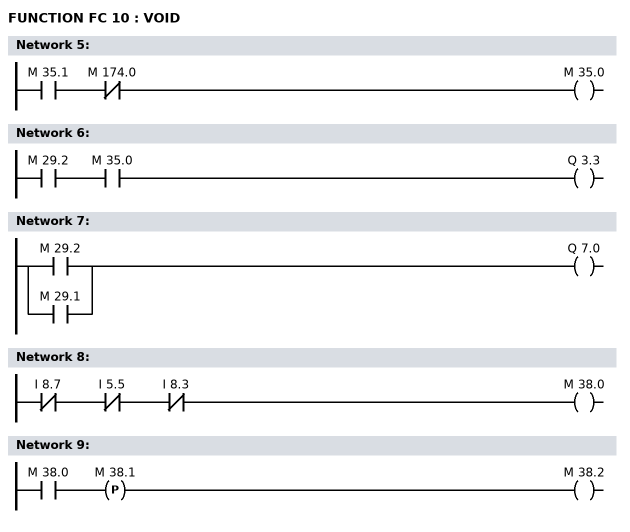

      A     M     35.1;
      AN    M    174.0;
      =     M     35.0;
NETWORK
TITLE =

      A     M     29.2;
      A     M     35.0;
      =     Q      3.3;
NETWORK
TITLE =

      O     M     29.2;
      O     M     29.1;
      =     Q      7.0;
NETWORK
TITLE =

      AN    I      8.7;
      AN    I      5.5;
      AN    I      8.3;
      =     M     38.0;
NETWORK
TITLE =

      A     M     38.0;
      FP    M     38.1;
      =     M     38.2;
NETWORK
TITLE =

      A     I      8.7;
      A(    ;
      A     I      5.5;
      L     DB2.DBW   46;
      SF    T     23;
      NOP   0;
      NOP   0;
      NOP   0;
      A     T     23;
      )     ;
      A     I      8.3;
      A     I     11.4;
      A     I     12.5;
      =     L      1.0;
      A     L      1.0;
      BLD   102;
      =     M     38.3;
      A     L      1.0;
      A     M     44.1;
      S     Q      3.5;
      A(    ;
      ON    M     44.1;
      O     ;
      A     I      0.6;
      AN    I      1.1;
      O     ;
      A     I      0.7;
      AN    I      4.1;
      )     ;
      R     Q      3.5;
      NOP   0;
NETWORK
TITLE =

      A(    ;
      A     M     35.0;
      A     #TEMP0;
      AN    #TEMP1;
      AN    M     38.3;
      FP    M     29.5;
      =     M     44.0;
      A     M     44.0;
      S     M     44.1;
      A(    ;
      O     M     20.7;
      ON    M     35.1;
      O     M     11.1;
      O     M     38.2;
      O     #TEMP1;
      O     M    114.0;
      )     ;
      R     M     44.1;
      A     M     44.1;
      )     ;
      A     M     38.3;
      O     ;
      AN    M     38.3;
      A     M     44.1;
      A     M     10.6;
      O     I      1.3;
      =     Q      3.1;
NETWORK
TITLE =
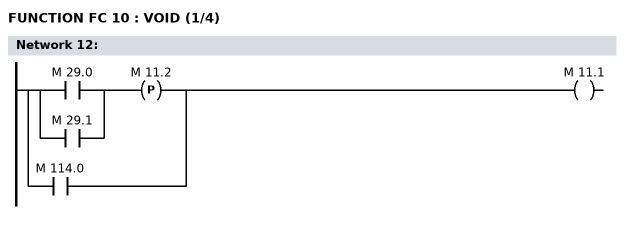

      A(    ;
      O     M     29.0;
      O     M     29.1;
      )     ;
      FP    M     11.2;
      O     M    114.0;
      =     M     11.1;
NETWORK
TITLE =
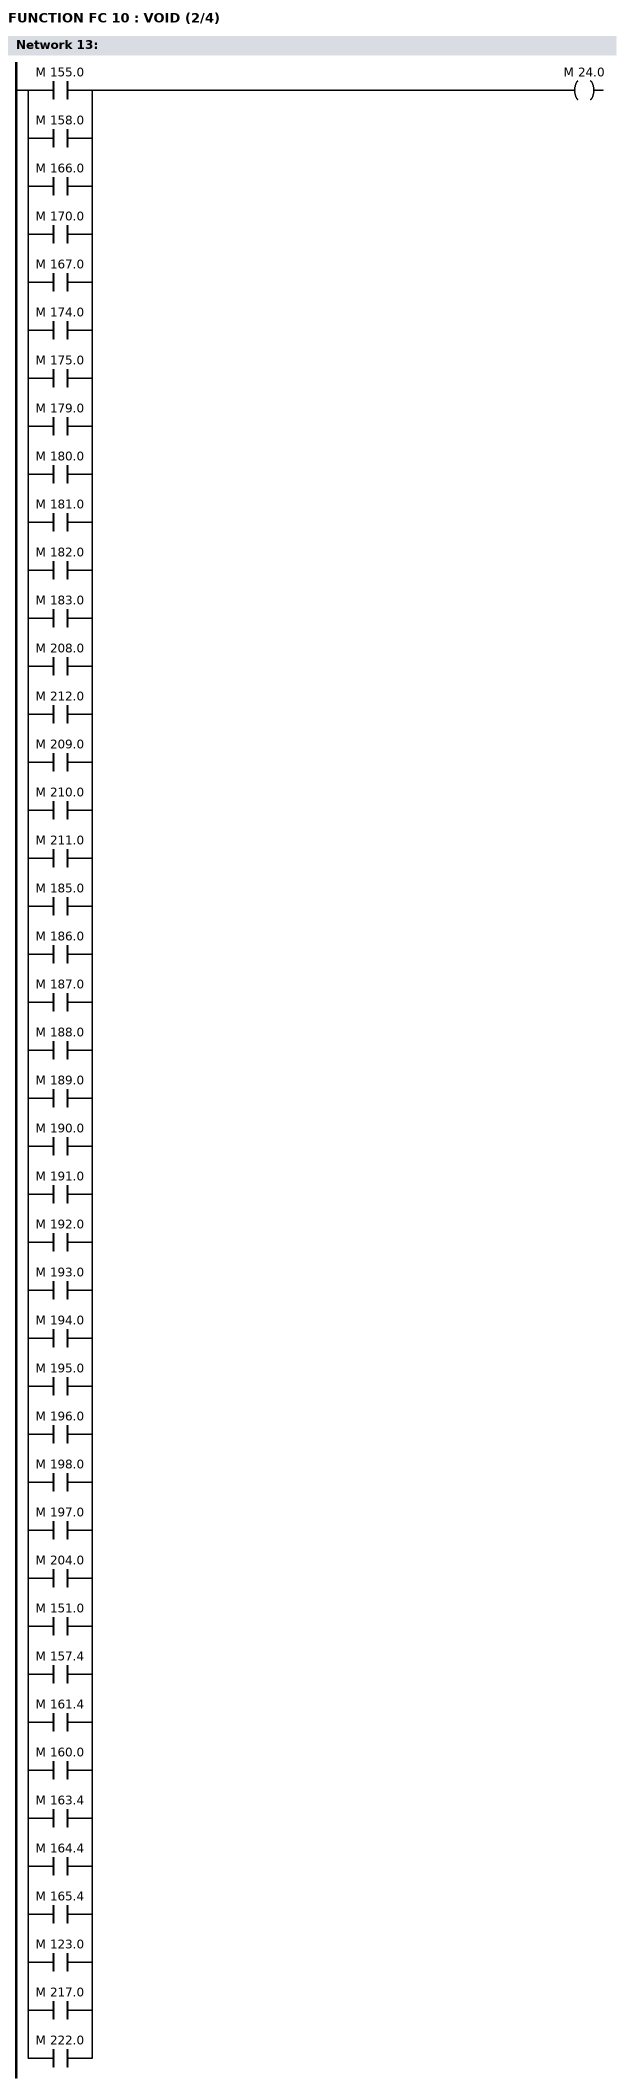

      O     M    155.0;
      O     M    158.0;
      O     M    166.0;
      O     M    170.0;
      O     M    167.0;
      O     M    174.0;
      O     M    175.0;
      O     M    179.0;
      O     M    180.0;
      O     M    181.0;
      O     M    182.0;
      O     M    183.0;
      O     M    208.0;
      O     M    212.0;
      O     M    209.0;
      O     M    210.0;
      O     M    211.0;
      O     M    185.0;
      O     M    186.0;
      O     M    187.0;
      O     M    188.0;
      O     M    189.0;
      O     M    190.0;
      O     M    191.0;
      O     M    192.0;
      O     M    193.0;
      O     M    194.0;
      O     M    195.0;
      O     M    196.0;
      O     M    198.0;
      O     M    197.0;
      O     M    204.0;
      O     M    151.0;
      O     M    157.4;
      O     M    161.4;
      O     M    160.0;
      O     M    163.4;
      O     M    164.4;
      O     M    165.4;
      O     M    123.0;
      O     M    217.0;
      O     M    222.0;
      =     M     24.0;
NETWORK
TITLE =
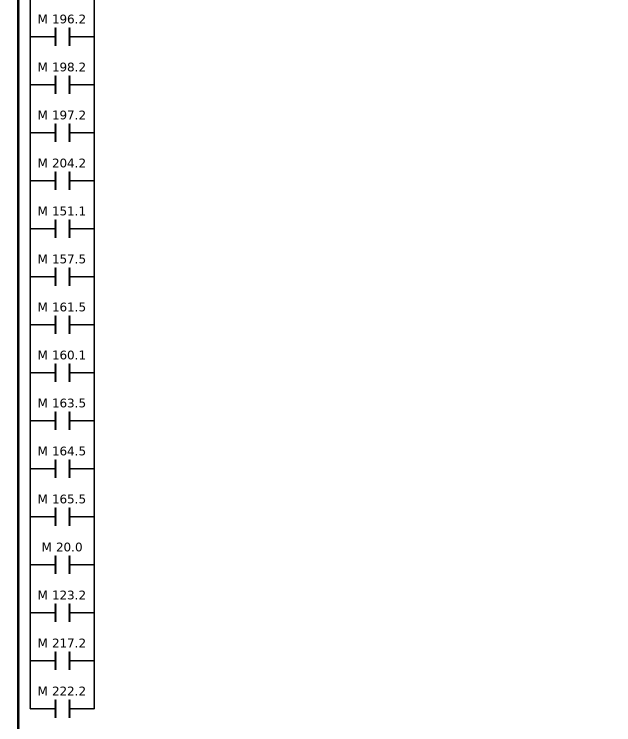

      O     M    155.2;
      O     M    158.2;
      O     M    166.2;
      O     M    170.2;
      O     M    167.2;
      O     M    174.2;
      O     M    175.2;
      O     M    179.2;
      O     M    180.2;
      O     M    181.2;
      O     M    182.2;
      O     M    183.2;
      O     M    208.2;
      O     M    212.2;
      O     M    209.2;
      O     M    210.2;
      O     M    211.2;
      O     M    185.2;
      O     M    186.2;
      O     M    187.2;
      O     M    188.2;
      O     M    189.2;
      O     M    190.2;
      O     M    191.2;
      O     M    192.2;
      O     M    193.2;
      O     M    194.2;
      O     M    195.2;
      O     M    196.2;
      O     M    198.2;
      O     M    197.2;
      O     M    204.2;
      O     M    151.1;
      O     M    157.5;
      O     M    161.5;
      O     M    160.1;
      O     M    163.5;
      O     M    164.5;
      O     M    165.5;
      O     M     20.0;
      O     M    123.2;
      O     M    217.2;
      O     M    222.2;
      =     M     22.0;
NETWORK
TITLE =
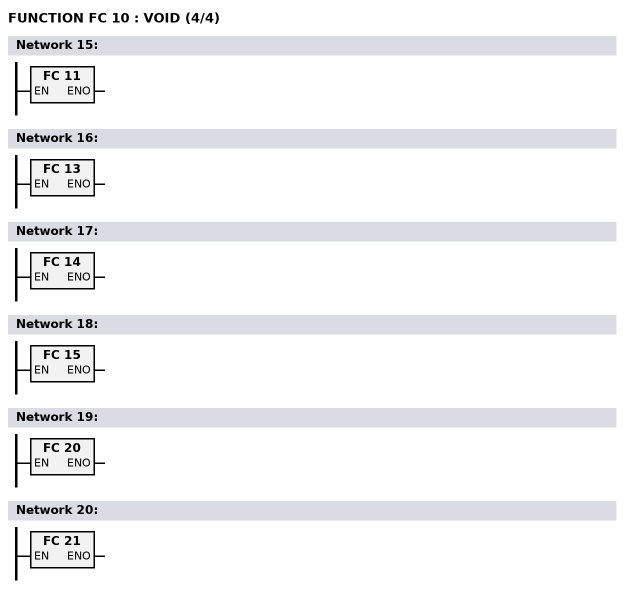

      CALL FC    11 ;
      NOP   0;
NETWORK
TITLE =

      CALL FC    13 ;
      NOP   0;
NETWORK
TITLE =

      CALL FC    14 ;
      NOP   0;
NETWORK
TITLE =

      CALL FC    15 ;
      NOP   0;
NETWORK
TITLE =

      CALL FC    20 ;
      NOP   0;
NETWORK
TITLE =

      CALL FC    21 ;
      NOP   0;
END_FUNCTION

FUNCTION FC 191 : VOID
AUTHOR :
FAMILY : ZEITEN
NAME : S_EVERZ
VERSION : 0.0


VAR_INPUT
  IN0 : BOOL ;
  IN1 : BOOL ;
END_VAR
VAR_IN_OUT
  IO2 : INT ;
  IO3 : INT ;
  IO4 : INT ;
  IO5 : INT ;
  IO6 : INT ;
  IO7 : WORD ;
END_VAR
VAR_TEMP
  TEMP8 : BOOL ;
  TEMP9 : BOOL ;
  TEMP10 : BOOL ;
  TEMP11 : BOOL ;
  TEMP12 : BOOL ;
END_VAR
BEGIN
NETWORK
TITLE =
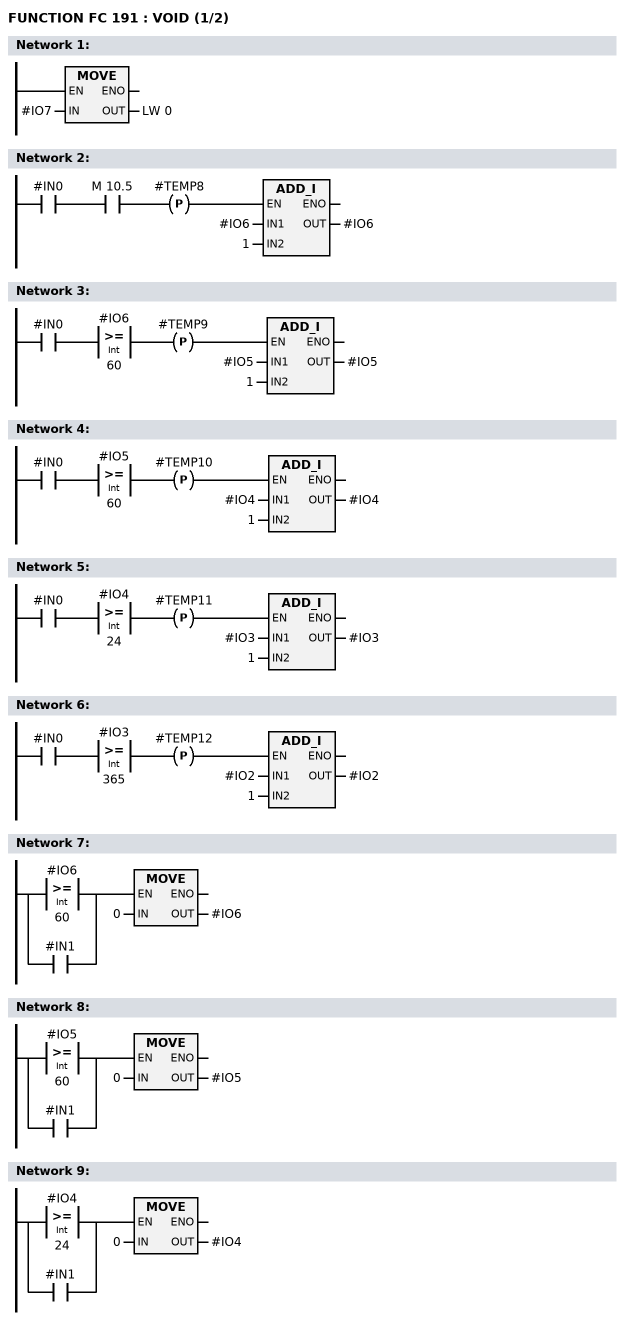

      L     #IO7;
      T     LW     0;
      NOP   0;
NETWORK
TITLE =

      A     #IN0;
      A     M     10.5;
      FP    #TEMP8;
      JNB   M001;
      L     #IO6;
      L     1;
      +I    ;
      T     #IO6;
M001: NOP   0;
NETWORK
TITLE =

      A     #IN0;
      A(    ;
      L     #IO6;
      L     60;
      >=I   ;
      )     ;
      FP    #TEMP9;
      JNB   M002;
      L     #IO5;
      L     1;
      +I    ;
      T     #IO5;
M002: NOP   0;
NETWORK
TITLE =

      A     #IN0;
      A(    ;
      L     #IO5;
      L     60;
      >=I   ;
      )     ;
      FP    #TEMP10;
      JNB   M003;
      L     #IO4;
      L     1;
      +I    ;
      T     #IO4;
M003: NOP   0;
NETWORK
TITLE =

      A     #IN0;
      A(    ;
      L     #IO4;
      L     24;
      >=I   ;
      )     ;
      FP    #TEMP11;
      JNB   M004;
      L     #IO3;
      L     1;
      +I    ;
      T     #IO3;
M004: NOP   0;
NETWORK
TITLE =

      A     #IN0;
      A(    ;
      L     #IO3;
      L     365;
      >=I   ;
      )     ;
      FP    #TEMP12;
      JNB   M005;
      L     #IO2;
      L     1;
      +I    ;
      T     #IO2;
M005: NOP   0;
NETWORK
TITLE =

      A(    ;
      O(    ;
      L     #IO6;
      L     60;
      >=I   ;
      )     ;
      O     #IN1;
      )     ;
      JNB   M006;
      L     0;
      T     #IO6;
M006: NOP   0;
NETWORK
TITLE =

      A(    ;
      O(    ;
      L     #IO5;
      L     60;
      >=I   ;
      )     ;
      O     #IN1;
      )     ;
      JNB   M007;
      L     0;
      T     #IO5;
M007: NOP   0;
NETWORK
TITLE =

      A(    ;
      O(    ;
      L     #IO4;
      L     24;
      >=I   ;
      )     ;
      O     #IN1;
      )     ;
      JNB   M008;
      L     0;
      T     #IO4;
M008: NOP   0;
NETWORK
TITLE =
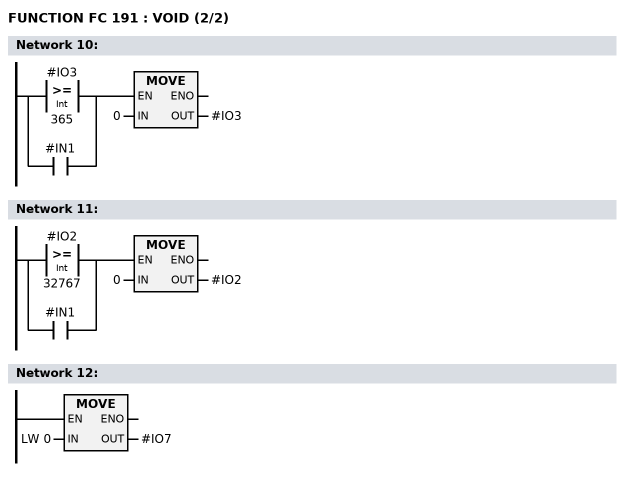

      A(    ;
      O(    ;
      L     #IO3;
      L     365;
      >=I   ;
      )     ;
      O     #IN1;
      )     ;
      JNB   M009;
      L     0;
      T     #IO3;
M009: NOP   0;
NETWORK
TITLE =

      A(    ;
      O(    ;
      L     #IO2;
      L     32767;
      >=I   ;
      )     ;
      O     #IN1;
      )     ;
      JNB   M00a;
      L     0;
      T     #IO2;
M00a: NOP   0;
NETWORK
TITLE =

      L     LW     0;
      T     #IO7;
      NOP   0;
END_FUNCTION

FUNCTION FC 1 : VOID
AUTHOR :
FAMILY : GENERAL
NAME : GENERAL
VERSION : 0.0

BEGIN
NETWORK
TITLE =
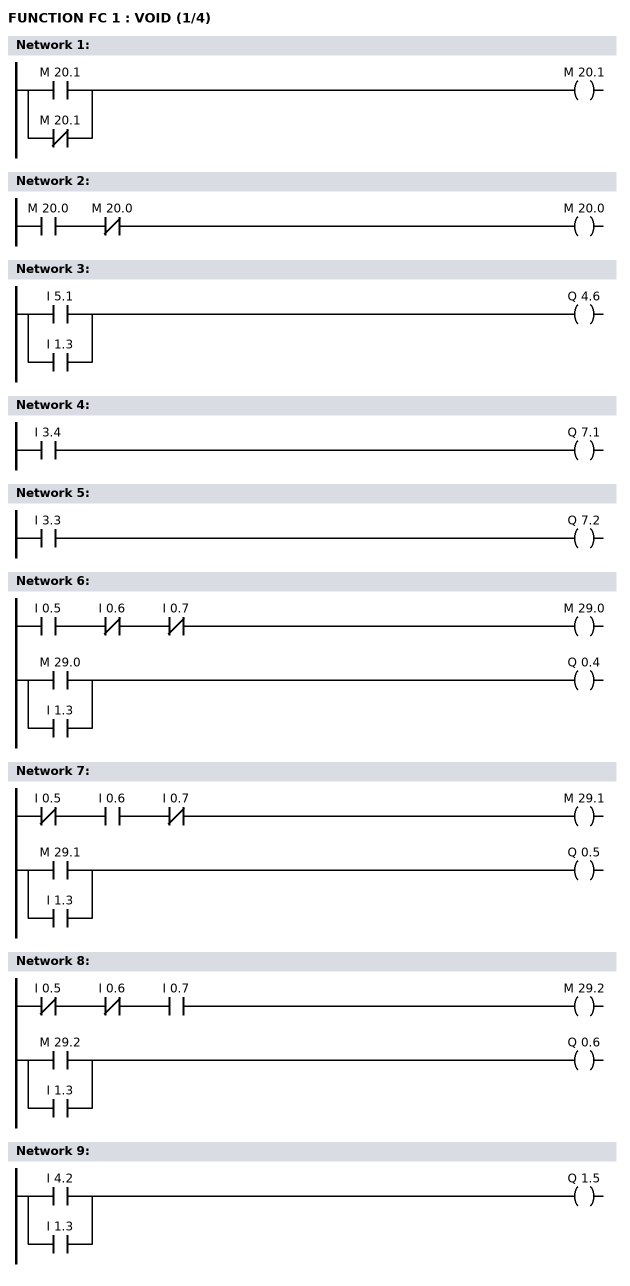

      O     M     20.1;
      ON    M     20.1;
      =     M     20.1;
NETWORK
TITLE =

      A     M     20.0;
      AN    M     20.0;
      =     M     20.0;
NETWORK
TITLE =

      O     I      5.1;
      O     I      1.3;
      =     Q      4.6;
NETWORK
TITLE =

      A     I      3.4;
      =     Q      7.1;
NETWORK
TITLE =

      A     I      3.3;
      =     Q      7.2;
NETWORK
TITLE =

      A     I      0.5;
      AN    I      0.6;
      AN    I      0.7;
      =     M     29.0;
      A     M     29.0;
      O     I      1.3;
      =     Q      0.4;
NETWORK
TITLE =

      AN    I      0.5;
      A     I      0.6;
      AN    I      0.7;
      =     M     29.1;
      A     M     29.1;
      O     I      1.3;
      =     Q      0.5;
NETWORK
TITLE =

      AN    I      0.5;
      AN    I      0.6;
      A     I      0.7;
      =     M     29.2;
      A     M     29.2;
      O     I      1.3;
      =     Q      0.6;
NETWORK
TITLE =

      O     I      4.2;
      O     I      1.3;
      =     Q      1.5;
NETWORK
TITLE =
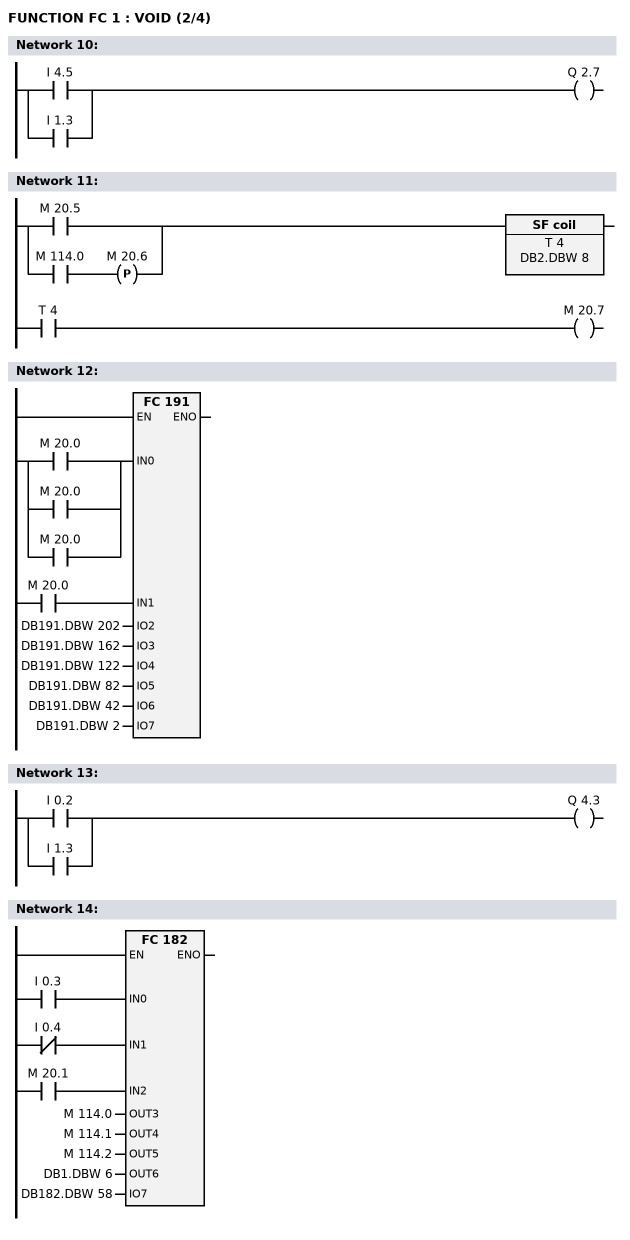

      O     I      4.5;
      O     I      1.3;
      =     Q      2.7;
NETWORK
TITLE =

      A(    ;
      O     M     20.5;
      O(    ;
      A     M    114.0;
      FP    M     20.6;
      )     ;
      )     ;
      L     DB2.DBW    8;
      SF    T      4;
      NOP   0;
      NOP   0;
      NOP   0;
      A     T      4;
      =     M     20.7;
NETWORK
TITLE =

      A(    ;
      O     M     20.0;
      O     M     20.0;
      O     M     20.0;
      )     ;
      =     L      0.0;
      BLD   103;
      A     M     20.0;
      =     L      0.1;
      BLD   103;
      CALL FC   191 (
           IN0                      := L      0.0,
           IN1                      := L      0.1,
           IO2                      := DB191.DBW  202,
           IO3                      := DB191.DBW  162,
           IO4                      := DB191.DBW  122,
           IO5                      := DB191.DBW   82,
           IO6                      := DB191.DBW   42,
           IO7                      := DB191.DBW    2);
      NOP   0;
NETWORK
TITLE =

      O     I      0.2;
      O     I      1.3;
      =     Q      4.3;
NETWORK
TITLE =

      A     I      0.3;
      =     L      0.0;
      BLD   103;
      AN    I      0.4;
      =     L      0.1;
      BLD   103;
      A     M     20.1;
      =     L      0.2;
      BLD   103;
      CALL FC   182 (
           IN0                      := L      0.0,
           IN1                      := L      0.1,
           IN2                      := L      0.2,
           OUT3                     := M    114.0,
           OUT4                     := M    114.1,
           OUT5                     := M    114.2,
           OUT6                     := DB1.DBW    6,
           IO7                      := DB182.DBW   58);
      NOP   0;
NETWORK
TITLE =
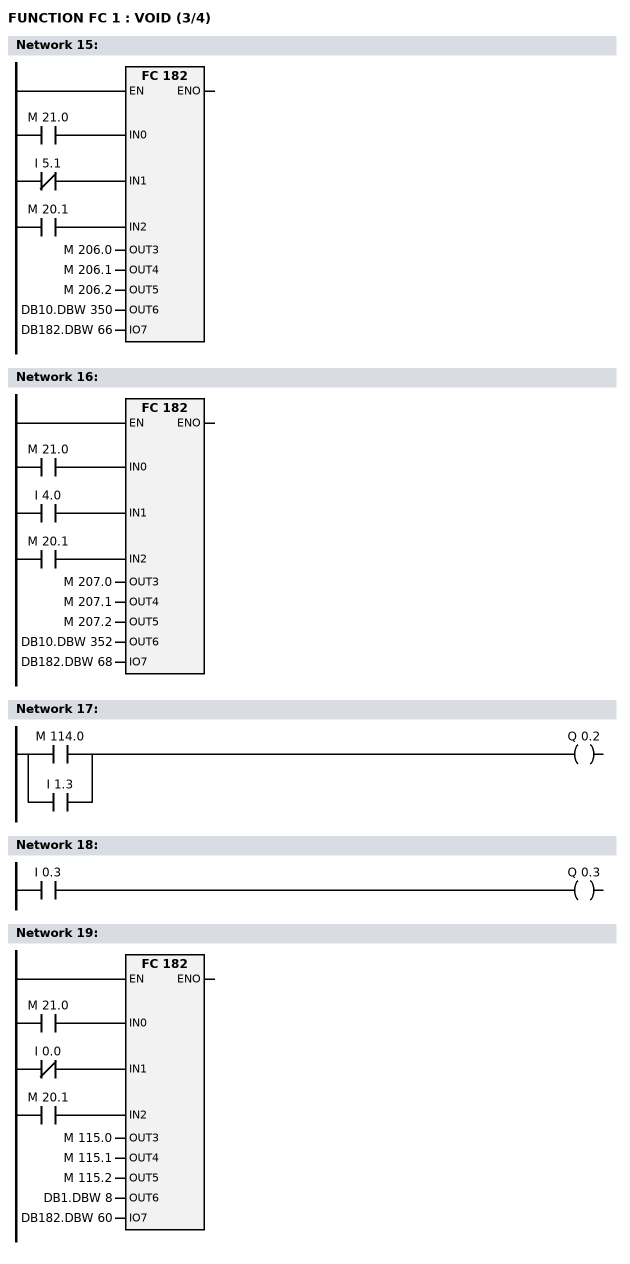

      A     M     21.0;
      =     L      0.0;
      BLD   103;
      AN    I      5.1;
      =     L      0.1;
      BLD   103;
      A     M     20.1;
      =     L      0.2;
      BLD   103;
      CALL FC   182 (
           IN0                      := L      0.0,
           IN1                      := L      0.1,
           IN2                      := L      0.2,
           OUT3                     := M    206.0,
           OUT4                     := M    206.1,
           OUT5                     := M    206.2,
           OUT6                     := DB10.DBW  350,
           IO7                      := DB182.DBW   66);
      NOP   0;
NETWORK
TITLE =

      A     M     21.0;
      =     L      0.0;
      BLD   103;
      A     I      4.0;
      =     L      0.1;
      BLD   103;
      A     M     20.1;
      =     L      0.2;
      BLD   103;
      CALL FC   182 (
           IN0                      := L      0.0,
           IN1                      := L      0.1,
           IN2                      := L      0.2,
           OUT3                     := M    207.0,
           OUT4                     := M    207.1,
           OUT5                     := M    207.2,
           OUT6                     := DB10.DBW  352,
           IO7                      := DB182.DBW   68);
      NOP   0;
NETWORK
TITLE =

      O     M    114.0;
      O     I      1.3;
      =     Q      0.2;
NETWORK
TITLE =

      A     I      0.3;
      =     Q      0.3;
NETWORK
TITLE =

      A     M     21.0;
      =     L      0.0;
      BLD   103;
      AN    I      0.0;
      =     L      0.1;
      BLD   103;
      A     M     20.1;
      =     L      0.2;
      BLD   103;
      CALL FC   182 (
           IN0                      := L      0.0,
           IN1                      := L      0.1,
           IN2                      := L      0.2,
           OUT3                     := M    115.0,
           OUT4                     := M    115.1,
           OUT5                     := M    115.2,
           OUT6                     := DB1.DBW    8,
           IO7                      := DB182.DBW   60);
      NOP   0;
NETWORK
TITLE =
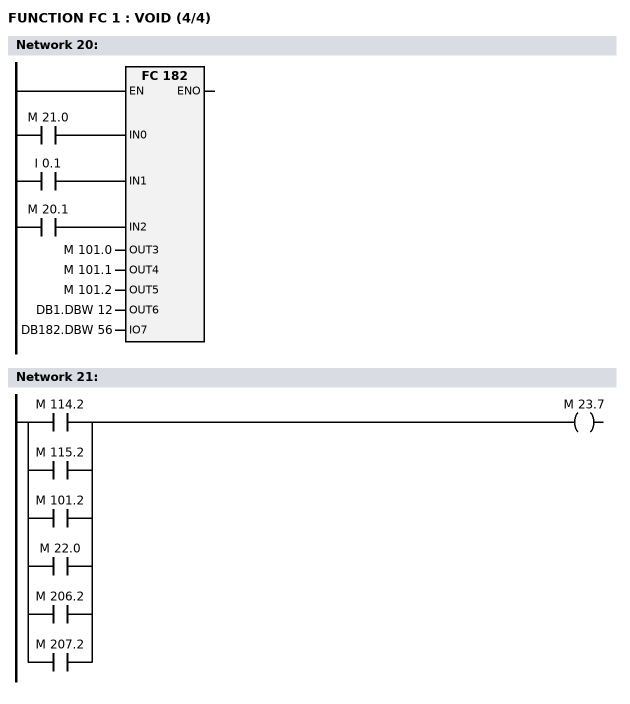

      A     M     21.0;
      =     L      0.0;
      BLD   103;
      A     I      0.1;
      =     L      0.1;
      BLD   103;
      A     M     20.1;
      =     L      0.2;
      BLD   103;
      CALL FC   182 (
           IN0                      := L      0.0,
           IN1                      := L      0.1,
           IN2                      := L      0.2,
           OUT3                     := M    101.0,
           OUT4                     := M    101.1,
           OUT5                     := M    101.2,
           OUT6                     := DB1.DBW   12,
           IO7                      := DB182.DBW   56);
      NOP   0;
NETWORK
TITLE =

      O     M    114.2;
      O     M    115.2;
      O     M    101.2;
      O     M     22.0;
      O     M    206.2;
      O     M    207.2;
      =     M     23.7;
NETWORK
TITLE =

      O     M    114.0;
      O     M    115.0;
      O     M    101.0;
      O     M     24.0;
      O     M    206.0;
      O     M    207.0;
      =     L      0.0;
      O     L      0.0;
      O     I      1.3;
      =     Q      1.0;
      A     L      0.0;
      BLD   102;
      =     Q      3.4;
NETWORK
TITLE =
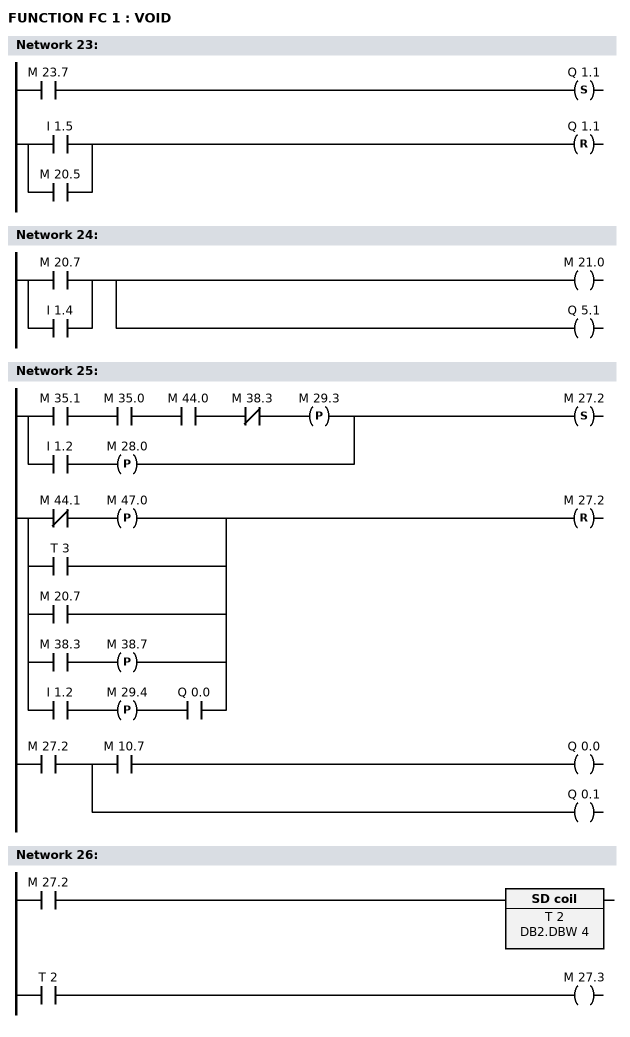

      A     M     23.7;
      S     Q      1.1;
      A(    ;
      O     I      1.5;
      O     M     20.5;
      )     ;
      R     Q      1.1;
      NOP   0;
NETWORK
TITLE =

      O     M     20.7;
      O     I      1.4;
      =     M     21.0;
      =     Q      5.1;
NETWORK
TITLE =

      A(    ;
      A     M     35.1;
      A     M     35.0;
      A     M     44.0;
      AN    M     38.3;
      FP    M     29.3;
      O(    ;
      A     I      1.2;
      FP    M     28.0;
      )     ;
      )     ;
      S     M     27.2;
      A(    ;
      AN    M     44.1;
      FP    M     47.0;
      O     T      3;
      O     M     20.7;
      O(    ;
      A     M     38.3;
      FP    M     38.7;
      )     ;
      O(    ;
      A     I      1.2;
      FP    M     29.4;
      A     Q      0.0;
      )     ;
      )     ;
      R     M     27.2;
      A     M     27.2;
      =     L      0.0;
      A     L      0.0;
      A     M     10.7;
      =     Q      0.0;
      A     L      0.0;
      BLD   102;
      =     Q      0.1;
NETWORK
TITLE =

      A     M     27.2;
      L     DB2.DBW    4;
      SD    T      2;
      NOP   0;
      NOP   0;
      NOP   0;
      A     T      2;
      =     M     27.3;
NETWORK
TITLE =

      A(    ;
      A     M     27.2;
      L     DB2.DBW   10;
      SD    T      5;
      NOP   0;
      NOP   0;
      NOP   0;
      A     T      5;
      )     ;
      L     DB2.DBW    6;
      SE    T      3;
      NOP   0;
      NOP   0;
      NOP   0;
      NOP   0;
NETWORK
TITLE =

      CALL FC     3 ;
      NOP   0;
NETWORK
TITLE =

      CALL FC    10 ;
      NOP   0;
END_FUNCTION

FUNCTION FC 186 : VOID
AUTHOR :
FAMILY : GENERAL
NAME : BYTECOMP
VERSION : 0.0


VAR_INPUT
  IN0 : BYTE ;
  IN1 : BYTE ;
END_VAR
VAR_OUTPUT
  OUT2 : BOOL ;
  OUT3 : BOOL ;
  OUT4 : BOOL ;
  OUT5 : BOOL ;
END_VAR
VAR_TEMP
  TEMP6 : INT ;
  TEMP7 : INT ;
END_VAR
BEGIN
NETWORK
TITLE =
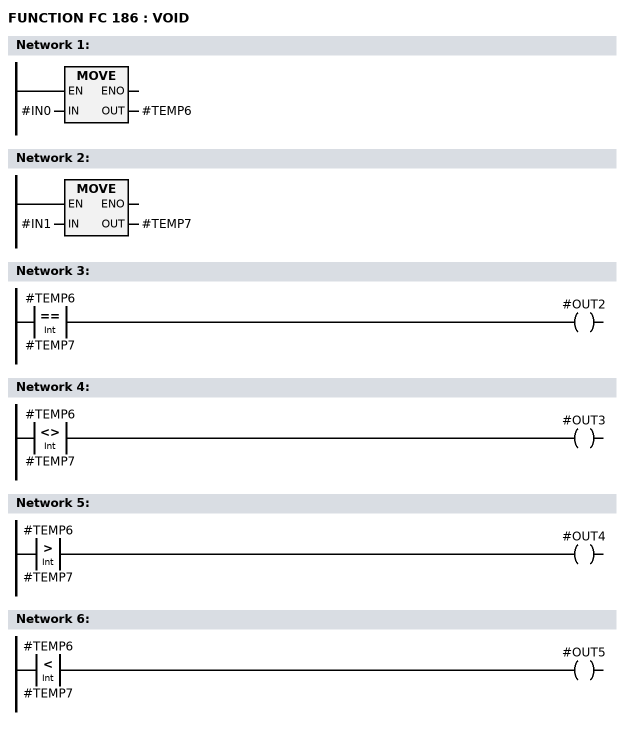

      L     #IN0;
      T     #TEMP6;
      NOP   0;
NETWORK
TITLE =

      L     #IN1;
      T     #TEMP7;
      NOP   0;
NETWORK
TITLE =

      L     #TEMP6;
      L     #TEMP7;
      ==I   ;
      =     #OUT2;
NETWORK
TITLE =

      L     #TEMP6;
      L     #TEMP7;
      <>I   ;
      =     #OUT3;
NETWORK
TITLE =

      L     #TEMP6;
      L     #TEMP7;
      >I    ;
      =     #OUT4;
NETWORK
TITLE =

      L     #TEMP6;
      L     #TEMP7;
      <I    ;
      =     #OUT5;
END_FUNCTION

ORGANIZATION_BLOCK OB 1
VERSION : 0.1


VAR_TEMP
  TEMP0 : BYTE ;
  TEMP1 : BYTE ;
  TEMP2 : BYTE ;
  TEMP3 : BYTE ;
  TEMP4 : BYTE ;
  TEMP5 : BYTE ;
  TEMP6 : INT ;
  TEMP7 : INT ;
  TEMP8 : INT ;
  TEMP9 : DATE_AND_TIME ;
  TEMP10 : WORD ;
END_VAR
BEGIN
NETWORK
TITLE =

      CALL FC   186 (
           IN0                      := #TEMP1,
           IN1                      := B#16#1,
           OUT2                     := M     20.5,
           OUT3                     := M     20.2,
           OUT4                     := M     20.2,
           OUT5                     := M     20.2);
      NOP   0;
NETWORK
TITLE =

      CALL FC     1 ;
      NOP   0;
END_ORGANIZATION_BLOCK

ORGANIZATION_BLOCK OB 85
VERSION : 0.0


VAR_TEMP
  TEMP0 : BYTE ;
  TEMP1 : BYTE ;
  TEMP2 : BYTE ;
  TEMP3 : BYTE ;
  TEMP4 : BYTE ;
  TEMP5 : BYTE ;
  TEMP6 : INT ;
  TEMP7 : BYTE ;
  TEMP8 : BYTE ;
  TEMP9 : BYTE ;
  TEMP10 : BYTE ;
  TEMP11 : DATE_AND_TIME ;
END_VAR
BEGIN
END_ORGANIZATION_BLOCK

ORGANIZATION_BLOCK OB 86
VERSION : 0.0


VAR_TEMP
  TEMP0 : BYTE ;
  TEMP1 : BYTE ;
  TEMP2 : BYTE ;
  TEMP3 : BYTE ;
  TEMP4 : BYTE ;
  TEMP5 : BYTE ;
  TEMP6 : WORD ;
  TEMP7 : ARRAY  [0 .. 31 ] OF BOOL ;
  TEMP8 : DATE_AND_TIME ;
END_VAR
BEGIN
END_ORGANIZATION_BLOCK

ORGANIZATION_BLOCK OB 122
VERSION : 0.0


VAR_TEMP
  TEMP0 : BYTE ;
  TEMP1 : BYTE ;
  TEMP2 : BYTE ;
  TEMP3 : BYTE ;
  TEMP4 : BYTE ;
  TEMP5 : BYTE ;
  TEMP6 : WORD ;
  TEMP7 : WORD ;
  TEMP8 : WORD ;
  TEMP9 : DATE_AND_TIME ;
END_VAR
BEGIN
END_ORGANIZATION_BLOCK

